FUNCTION_BLOCK CAT1_HMI (* Service Interface Function Block Type *)
  (* Standard: 61499-2 *)
  (* Version 0.0, 22/06/2021, Pranay Jhunjhunwala, Schneider Electric, template *)
  PACKAGE Main;
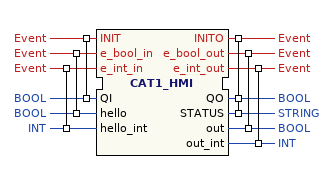
  EVENT_INPUT
    INIT WITH QI;
    e_bool_in WITH hello;
    e_int_in WITH hello_int;
  END_EVENT
  EVENT_OUTPUT
    INITO WITH QO, STATUS;
    e_bool_out WITH out;
    e_int_out WITH out_int;
  END_EVENT
  VAR_INPUT
    QI : BOOL;
    hello : BOOL;
    hello_int : INT;
  END_VAR
  VAR_OUTPUT
    QO : BOOL; (* Event Output Qualifier *)
    STATUS : STRING; (* Service Status *)
    out : BOOL;
    out_int : INT;
  END_VAR
  SERVICE /
    SEQUENCE 
    END_SEQUENCE
  END_SERVICE
END_FUNCTION_BLOCK
